Yaskawa INFORM job: valve_planes_program.JBI

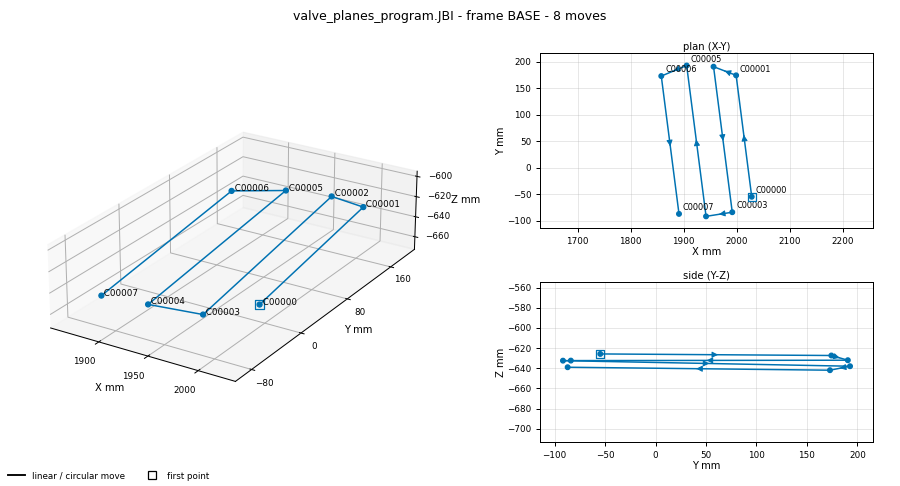
[picture p0: tool path of valve_planes_program.JBI in frame BASE, 8 of 10 moves have a stored position in this frame; points joined in program order, loops and branches not executed]
/JOB
//NAME valve_planes_program
//POS
///NPOS 8,0,8,0,0,0
///TOOL 0
///POSTYPE BASE
///RECTAN
///RCONF 0,0,0,0,0,0,0,0,0,0,0,0,0,0,0,0,0,0,0,0,0,0,0,0
C00000=2028.128418,-54.745615,-625.778350,-175.000000,-7.965706,-5.000000
C00001=1998.692475,174.205975,-627.333321,-175.000000,-7.965706,-5.000000
C00002=1956.151836,190.504300,-631.989321,-175.000000,-7.965706,-5.000000
C00003=1991.431902,-83.902644,-632.380321,-175.000000,-7.965706,-5.000000
C00004=1942.022561,-91.697803,-632.444321,-175.000000,-7.965706,-5.000000
C00005=1905.460052,192.683939,-637.947321,-175.000000,-7.965706,-5.000000
C00006=1857.588005,172.814139,-641.896321,-175.000000,-7.965706,-5.000000
C00007=1891.000073,-87.063596,-638.950321,-175.000000,-7.965706,-5.000000
///POSTYPE PULSE
///PULSE
EC00000=7168.0
EC00001=7168.0
EC00002=7168.0
EC00003=7168.0
EC00004=7168.0
EC00005=7168.0
EC00006=7168.0
EC00007=7168.0
//INST
///DATE 2023/08/16 18:06
///ATTR SC,RW,RJ
////FRAME BASE
///GROUP1 RB1,ST1
NOP
MOVJ P009 EX000 VJ=15.00
MOVJ C00000 EC00000 VJ=15.0
CALL JOB:SPYON
MOVL C00001 EC00001 V=150.0
MOVL C00002 EC00002 V=150.0
MOVL C00003 EC00003 V=150.0
MOVL C00004 EC00004 V=150.0
MOVL C00005 EC00005 V=150.0
MOVL C00006 EC00006 V=150.0
MOVL C00007 EC00007 V=150.0
CALL JOB:SPYOF
MOVJ P009 VJ=15.00
END
